FUNCTION F_VerifyAllTransportTubeStatuses : BOOL
VAR_INPUT
	stExpStatus : ST_TransportTubeStatuses;
	stStatusOp : ST_TransportTubeOps;
	bEnforce : BOOL;
END_VAR
VAR
	nIter : UINT;
	bResult : BOOL := TRUE;
END_VAR

FOR nIter := 1 TO GVL_TransportTubes.NUM_TRANSPORT_TUBES DO
	bResult := bResult AND F_VerifyTransportTubeStatuses(
		stExpStatus := stExpStatus,
		stStatusOp := stStatusOp,
		eTransportTube := GVL_TransportTubes.aTubes[nIter],
		bEnforce := bEnforce);
END_FOR

F_VerifyAllTransportTubeStatuses := bResult;

END_FUNCTION

(* stored: Version 1.1.0.1, ProductVersion 3.1.4024.0
   POU F_VerifyAllTransportTubeStatuses: Id {358b5524-2bc6-4c0c-884c-f5fe5398d76e}, SpecialFunc None *)
